Yaskawa INFORM job: TEST-S2-SAFETY.JBI

/JOB
//NAME TEST-S2-SAFETY
//POS
///NPOS 0,0,0,0,0,1
///TOOL 0
///POSTYPE ANGLE
///ANGLE
EX00000=0.0000
//INST
///DATE 2018/11/13 14:18
///ATTR SC,RW
///GROUP1 ST2
NOP
MOVJ EX000 VJ=100.00
MOVJ EX000 VJ=100.00
END
